(* PLC project cb_tof, Dassault Systèmes ControlBuild 2024x *)
(* stored: creationDateTime 2023-10-03T11:12:44-01:00 *)

(* This is a IEC 1131-3 TOFF Timer *)
FUNCTION_BLOCK timers_counters.cb_tof
  VAR_INPUT
    IN : BOOL := false;
    PT : TIME := T#0h0m0s0ms;
  END_VAR
  VAR_OUTPUT
    Q0 : BOOL := false;
    CV : TIME := T#0h0m0s0ms;
  END_VAR
  VAR
    memo_tof : BOOL := false;
  END_VAR


ACTION C_source_code:
/* -----------------------------------------------------------------	*/
/* Type : BFU									*/
/* Copyright : Geensoft							*/
/* Version : 1.1 23/03/2010							*/
/* -----------------------------------------------------------------	*/
/* This is a Timing upon de-activation  (TOF)				*/
/* -------------------------------------------------------------	*/

	double PT_double;
	double v_t1;		// value temporary clocks in tenth of milliseconds
	double v_nbDays_t1;

	//calculation of the duration in tenth of milliseconds (number of days included)
	v_t1 = CV(1)*24.0*3600.0*10000.0 + CV(2);

	//calculation of the duration in tenth of milliseconds (number of days included)
	PT_double = PT(1)*24.0*3600.0*10000.0 + PT(2);

	if((PT_double < 0) || (PT_double > 9223372036854775807.0)) {
		memo_tof=0;
		CV(1) = CV(2) = 0;
		Q0 = 0;
	}
	else {
		if(IN) {
			v_t1 = 0.0;
			memo_tof = 1;
		}
		else {
			if (memo_tof == 1) {
				v_t1 = v_t1 + (CLOCK_PERIOD / 100.0);
			};
			if (v_t1 > PT_double) {
				v_t1 = PT_double;
				memo_tof = 0;
			}
		}
		//conversion of temporary clocks in a time format
		modf(v_t1/(24.0*3600.0*10000.0), &v_nbDays_t1);
		CV(2) = (long) v_t1 - v_nbDays_t1*24.0*3600.0*10000.0;
		CV(1) = (long) v_nbDays_t1;
		if (PT_double==0.0) {
			Q0=0;
		}
		else {
			Q0 = (v_t1 <= PT_double) && (memo_tof == 1);
		}
	}
END_ACTION

ACTION C_header:
//#include "cb_memory.h"
END_ACTION
END_FUNCTION_BLOCK
